TYPE WcStateBase_A2171C4E :
STRUCT
END_STRUCT
END_TYPE

(* stored: Version 1.2.0.0, ProductVersion 3.1.4024.9
   DUT WcStateBase_A2171C4E: Id {f733ca8a-99a9-4ac7-a35b-a2236ba3e99d} *)
